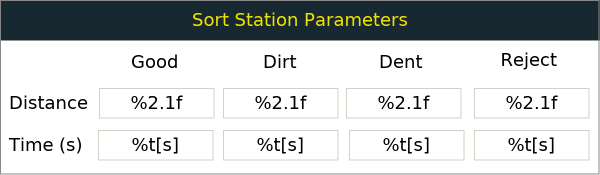
VISUALIZATION AOISortStationFrame  // 600x175
    Rectangle (0,0 600x40), "Sort Station Parameters"
    Label (6,130 90x30), "Time (s)"
    Label (6,88 90x30), "Distance"
    Label (110,47 90x30), "Good"
    Label (235,47 90x30), "Dirt"
    Label (356,47 90x30), "Dent"
    Label (484,45 90x30), "Reject"
    Textfield (99,88 115x30), "%2.1f", text variable: PRG_MachineControl.fbMachineControler.lrSortGoodDistance
        OnMouseClick: write the text variable via VisuDialogs.Numpad
    Textfield (223,88 115x30), "%2.1f", text variable: PRG_MachineControl.fbMachineControler.lrSortDirtDistance
        OnMouseClick: write the text variable via VisuDialogs.Numpad
    Textfield (346,88 115x30), "%2.1f", text variable: PRG_MachineControl.fbMachineControler.lrSortDentDistance
        OnMouseClick: write the text variable via VisuDialogs.Numpad
    Textfield (474,88 115x30), "%2.1f", text variable: PRG_MachineControl.fbMachineControler.lrSortRejectDistance
        OnMouseClick: write the text variable via VisuDialogs.Numpad
    Textfield (98,130 115x30), "%t[s]", text variable: PRG_MachineControl.fbMachineControler.tSortValveGoodTime
        OnMouseClick: write the text variable via VisuDialogs.Numpad
    Textfield (223,130 115x30), "%t[s]", text variable: PRG_MachineControl.fbMachineControler.tSortValveDirtTime
        OnMouseClick: write the text variable via VisuDialogs.Numpad
    Textfield (349,130 115x30), "%t[s]", text variable: PRG_MachineControl.fbMachineControler.tSortValveDentTime
        OnMouseClick: write the text variable via VisuDialogs.Numpad
    Textfield (474,130 115x30), "%t[s]", text variable: PRG_MachineControl.fbMachineControler.tSortValveRejectTime
        OnMouseClick: write the text variable via VisuDialogs.Numpad
END_VISUALIZATION

(* stored: Version 1.1.0.1, ProductVersion 3.1.4024.9
   Visu AOISortStationFrame: Id {7c771210-d44d-4f52-898c-7dd9dc66fee0} *)
